FUNCTION_BLOCK FB_MotionStageSim
(*
    Set all the values needed for a fake motor to be movable
    via the IOC, then call FB_MotionStage
*)
VAR_IN_OUT
    stMotionStage: ST_MotionStage;
END_VAR
VAR_INPUT
    nEnableMode: ENUM_StageEnableMode := ENUM_StageEnableMode.ALWAYS;
END_VAR
VAR
    fbMotionStage: FB_MotionStage;
    bInit: BOOL;
END_VAR

IF NOT bInit THEN
    bInit := TRUE;
    // Stand-in for no forward limit
    stMotionStage.bLimitForwardEnable := TRUE;
    // Stand-in for no reverse limit
    stMotionStage.bLimitBackwardEnable := TRUE;
    // Stand-in for no STO button
    stMotionStage.bHardwareEnable := TRUE;
    // Stand-in for no PMPS governer
    stMotionStage.bPowerSelf := TRUE;
    // Always keep it enabled for testing ease
    stMotionStage.nEnableMode := nEnableMode;
END_IF
// Call FB_MotionStage to do the thing
fbMotionStage(stMotionStage := stMotionStage);

END_FUNCTION_BLOCK

(* stored: Version 1.1.0.1, ProductVersion 3.1.4022.18
   POU FB_MotionStageSim: Id {d9a67e97-6cca-43d0-9ed9-24a1d18bbca1}, SpecialFunc None *)
